{attribute 'qualified_only'}
{attribute 'strict'}
TYPE eSupervisoryTransitions :
(
	create := 0,
	configure := 1,
	cleanup := 2,
	activate := 3,
	deactivate := 4,
	shutdown := 5,
	destroy := 6
);
END_TYPE

(* stored: Version 1.1.0.1, ProductVersion 3.1.4026.18
   DUT eSupervisoryTransitions: Id {a1b2c3d4-4444-4444-4444-444444444444} *)
